(* IEC 61131-3 sources: teller/JD_Teller_LC2_V11/Class/Machine_Settings, 1 file *)

(* ---- Machine_Settings.st ---- *)
(*!
<Class
	Name               = "Machine_Settings"
	Revision           = "1.5"
	RealtimeTask       = "false"
	CyclicTask         = "false"
	BackgroundTask     = "false"
	DefBackground      = "100 ms"
	Sigmatek           = "false"
	OSInterface        = "false"
	HighPriority       = "false"
	Automatic          = "false"
	UpdateMode         = "Prescan"
	SharedCommandTable = "true"
	Objectsize         = "(750,1620)">
	<Channels>
		<Server Name="ClassSvr" Visualized="false" Initialize="false" WriteProtected="true" Retentive="false"/>
		<Server Name="Comp_FreeJam" Visualized="true" Initialize="false" WriteProtected="false" Retentive="false"/>
		<Server Name="Comp_JamTeachIn" Visualized="true" Initialize="false" WriteProtected="false" Retentive="false"/>
		<Server Name="Comp_Teller" Visualized="true" Initialize="false" WriteProtected="false" Retentive="false"/>
		<Server Name="Comp_Teller_Menu" Visualized="true" Initialize="false" WriteProtected="false" Retentive="false"/>
		<Server Name="Comp_Ventieldriver" Visualized="true" Initialize="false" WriteProtected="false" Retentive="false"/>
		<Server Name="Opt_Operator_Login" Visualized="true" Initialize="false" WriteProtected="false" Retentive="false"/>
		<Server Name="Section_View_Rotate" Visualized="true" Initialize="false" WriteProtected="false" Retentive="false"/>
		<Client Name="cComp_FreeJam" Required="false" Internal="false"/>
		<Client Name="cComp_JamTeachIn" Required="false" Internal="false"/>
		<Client Name="cComp_Teller" Required="false" Internal="false"/>
		<Client Name="cComp_Ventieldriver" Required="true" Internal="false"/>
		<Client Name="cOpt_Operator_Login" Required="true" Internal="false"/>
		<Client Name="rComp_Bovenhaak1" Required="true" Internal="true"/>
		<Client Name="rComp_BoxEditor" Required="true" Internal="true"/>
		<Client Name="rComp_Feeder" Required="true" Internal="true"/>
		<Client Name="rComp_FreeJam" Required="true" Internal="true"/>
		<Client Name="rComp_Glue" Required="true" Internal="true"/>
		<Client Name="rComp_Haak1" Required="true" Internal="true"/>
		<Client Name="rComp_Haak2" Required="true" Internal="true"/>
		<Client Name="rComp_Haak3" Required="true" Internal="true"/>
		<Client Name="rComp_JamTeachIn" Required="true" Internal="true"/>
		<Client Name="rComp_RotStop" Required="true" Internal="true"/>
		<Client Name="rComp_Teller" Required="true" Internal="true"/>
		<Client Name="rComp_Ventieldriver" Required="true" Internal="true"/>
		<Client Name="rComp_Voorvouwhaak1" Required="true" Internal="true"/>
		<Client Name="rComp_Voorvouwhaak2" Required="true" Internal="true"/>
		<Client Name="rComp_Vouwriemregeling" Required="true" Internal="true"/>
		<Client Name="rOpt_Operator_Login" Required="true" Internal="true"/>
		<Client Name="rSection_ASection" Required="true" Internal="true"/>
		<Client Name="rSection_BSection" Required="true" Internal="true"/>
		<Client Name="rSection_Conveyor" Required="true" Internal="true"/>
		<Client Name="rSection_CSection" Required="true" Internal="true"/>
		<Client Name="rSection_Feeder" Required="true" Internal="true"/>
		<Client Name="rSection_FinalFold" Required="true" Internal="true"/>
		<Client Name="rSection_FUnit" Required="true" Internal="true"/>
		<Client Name="rSection_MAS" Required="true" Internal="true"/>
		<Client Name="rSection_PreFeeder" Required="true" Internal="true"/>
		<Client Name="rSection_Prefold" Required="true" Internal="true"/>
		<Client Name="rSection_TriFeeder" Required="true" Internal="true"/>
		<Client Name="rSection_Trombone" Required="true" Internal="true"/>
		<Client Name="rSection_View_Rotate" Required="true" Internal="true"/>
	</Channels>
	<RevDoku>
		<Owner Company="JD" Author="JVD"/>
		<Dokumentation Revision="1.5" Date="2014-01-27" Author="JVD" Company="JD" Description="ventieldrivers&#13;&#10;"/>
		<Dokumentation Revision="1.4" Date="2013-06-21" Author="JVD" Company="JD" Description="Extra server voor VVH2 toegevoegd&#13;&#10;"/>
		<Dokumentation Revision="1.3&#13;&#10;" Date="2012-03-28" Author="JVD" Company="JD" Description="Extra server voor de Voorvouwhaak toegevoegd&#13;&#10;"/>
		<Dokumentation Revision="1.2" Date="2011-12-08" Author="JVD" Company="JD" Description="-De servers werden Retentive gemaakt en via SRAM opgeslagen. Af en toe leverde dit problemen op waardoor waarders&#13;&#10;verloren zijn gegaan.&#13;&#10;Dit is opgelost door het gebruikt van Ram classjes in onderliggend netwerk. Peter van Oostrom heeft dit probleem onderkent.&#13;&#10;"/>
		<Dokumentation Revision="1.1" Date="2011-12-06" Author="JVD" Company="JD" Description="De autoSet instellingen zijn toegevoegd"/>
		<Dokumentation Revision="1.0" Date="2011-10-11" Author="JVD" Company="JD" Description="De Server Comp_Freejam toegevoegd"/>
	</RevDoku>
	<Network Name="Machine_Settings">
		<!-- List of Components in this network -->
		<Components>
			<Object
				Name       = "rComp_Bovenhaak1"
				Class      = "Ram"
				Position   = "(180,1620)"
				Visualized = "true">
				<Channels>
					<Server Name="Data"/>
				</Channels>
			</Object>
			<Object
				Name       = "rComp_BoxEditor"
				Class      = "Ram"
				Position   = "(180,180)"
				Visualized = "true">
				<Channels>
					<Server Name="Data"/>
				</Channels>
			</Object>
			<Object
				Name       = "rComp_Feeder"
				Class      = "Ram"
				Position   = "(180,900)"
				Visualized = "true">
				<Channels>
					<Server Name="Data"/>
				</Channels>
			</Object>
			<Object
				Name       = "rComp_FreeJam"
				Class      = "Ram"
				Position   = "(180,1800)"
				Visualized = "true">
				<Channels>
					<Server Name="Data"/>
				</Channels>
			</Object>
			<Object
				Name       = "rComp_Glue"
				Class      = "Ram"
				Position   = "(180,360)"
				Visualized = "true">
				<Channels>
					<Server Name="Data"/>
				</Channels>
			</Object>
			<Object
				Name       = "rComp_Haak1"
				Class      = "Ram"
				Position   = "(180,1080)"
				Visualized = "true">
				<Channels>
					<Server Name="Data"/>
				</Channels>
			</Object>
			<Object
				Name       = "rComp_Haak2"
				Class      = "Ram"
				Position   = "(180,1260)"
				Visualized = "true">
				<Channels>
					<Server Name="Data"/>
				</Channels>
			</Object>
			<Object
				Name       = "rComp_Haak3"
				Class      = "Ram"
				Position   = "(180,1440)"
				Visualized = "true">
				<Channels>
					<Server Name="Data"/>
				</Channels>
			</Object>
			<Object
				Name       = "rComp_JamTeachIn"
				Class      = "Ram"
				Position   = "(600,2160)"
				Visualized = "true">
				<Channels>
					<Server Name="Data"/>
				</Channels>
			</Object>
			<Object
				Name       = "rComp_RotStop"
				Class      = "Ram"
				Position   = "(180,720)"
				Visualized = "true">
				<Channels>
					<Server Name="Data"/>
				</Channels>
			</Object>
			<Object
				Name       = "rComp_Teller"
				Class      = "Ram"
				Position   = "(180,540)"
				Visualized = "true">
				<Channels>
					<Server Name="Data"/>
				</Channels>
			</Object>
			<Object
				Name       = "rComp_Ventieldriver"
				Class      = "Ram"
				Position   = "(180,2520)"
				Visualized = "true">
				<Channels>
					<Server Name="Data"/>
				</Channels>
			</Object>
			<Object
				Name       = "rComp_Voorvouwhaak1"
				Class      = "Ram"
				Position   = "(600,1980)"
				Visualized = "true">
				<Channels>
					<Server Name="Data"/>
				</Channels>
			</Object>
			<Object
				Name       = "rComp_Voorvouwhaak2"
				Class      = "Ram"
				Position   = "(600,2520)"
				Visualized = "true">
				<Channels>
					<Server Name="Data"/>
				</Channels>
			</Object>
			<Object
				Name       = "rComp_Vouwriemregeling"
				Class      = "Ram"
				Position   = "(600,2340)"
				Visualized = "true">
				<Channels>
					<Server Name="Data"/>
				</Channels>
			</Object>
			<Object
				Name       = "rOpt_Operator_Login"
				Class      = "Ram"
				Position   = "(180,2700)"
				Visualized = "true">
				<Channels>
					<Server Name="Data"/>
				</Channels>
			</Object>
			<Object
				Name       = "rSection_ASection"
				Class      = "Ram"
				Position   = "(600,540)"
				Visualized = "true">
				<Channels>
					<Server Name="Data"/>
				</Channels>
			</Object>
			<Object
				Name       = "rSection_BSection"
				Class      = "Ram"
				Position   = "(600,720)"
				Visualized = "true">
				<Channels>
					<Server Name="Data"/>
				</Channels>
			</Object>
			<Object
				Name       = "rSection_Conveyor"
				Class      = "Ram"
				Position   = "(600,1620)"
				Visualized = "true">
				<Channels>
					<Server Name="Data"/>
				</Channels>
			</Object>
			<Object
				Name       = "rSection_CSection"
				Class      = "Ram"
				Position   = "(600,900)"
				Visualized = "true">
				<Channels>
					<Server Name="Data"/>
				</Channels>
			</Object>
			<Object
				Name       = "rSection_Feeder"
				Class      = "Ram"
				Position   = "(180,1980)"
				Visualized = "true">
				<Channels>
					<Server Name="Data"/>
				</Channels>
			</Object>
			<Object
				Name       = "rSection_FinalFold"
				Class      = "Ram"
				Position   = "(600,1080)"
				Visualized = "true">
				<Channels>
					<Server Name="Data"/>
				</Channels>
			</Object>
			<Object
				Name       = "rSection_FUnit"
				Class      = "Ram"
				Position   = "(600,1260)"
				Visualized = "true">
				<Channels>
					<Server Name="Data"/>
				</Channels>
			</Object>
			<Object
				Name       = "rSection_MAS"
				Class      = "Ram"
				Position   = "(600,180)"
				Visualized = "true">
				<Channels>
					<Server Name="Data"/>
				</Channels>
			</Object>
			<Object
				Name       = "rSection_PreFeeder"
				Class      = "Ram"
				Position   = "(180,2160)"
				Visualized = "true">
				<Channels>
					<Server Name="Data"/>
				</Channels>
			</Object>
			<Object
				Name       = "rSection_Prefold"
				Class      = "Ram"
				Position   = "(600,360)"
				Visualized = "true">
				<Channels>
					<Server Name="Data"/>
				</Channels>
			</Object>
			<Object
				Name       = "rSection_TriFeeder"
				Class      = "Ram"
				Position   = "(180,2340)"
				Visualized = "true">
				<Channels>
					<Server Name="Data"/>
				</Channels>
			</Object>
			<Object
				Name       = "rSection_Trombone"
				Class      = "Ram"
				Position   = "(600,1440)"
				Visualized = "true">
				<Channels>
					<Server Name="Data"/>
				</Channels>
			</Object>
			<Object
				Name       = "rSection_View_Rotate"
				Class      = "Ram"
				Position   = "(600,1800)"
				Visualized = "true">
				<Channels>
					<Server Name="Data"/>
				</Channels>
			</Object>
		</Components>
		<Comments>
		</Comments>
		<!-- List of Connections in this network -->
		<Connections>
			<Connection Source="this.rComp_BoxEditor" Destination="rComp_BoxEditor.Data"/>
			<Connection Source="this.rComp_Glue" Destination="rComp_Glue.Data"/>
			<Connection Source="this.rComp_Teller" Destination="rComp_Teller.Data"/>
			<Connection Source="this.rComp_RotStop" Destination="rComp_RotStop.Data"/>
			<Connection Source="this.rComp_Feeder" Destination="rComp_Feeder.Data"/>
			<Connection Source="this.rComp_JamTeachIn" Destination="rComp_JamTeachIn.Data"/>
			<Connection Source="this.rComp_Haak1" Destination="rComp_Haak1.Data"/>
			<Connection Source="this.rComp_Haak2" Destination="rComp_Haak2.Data"/>
			<Connection Source="this.rComp_Haak3" Destination="rComp_Haak3.Data"/>
			<Connection Source="this.rComp_Bovenhaak1" Destination="rComp_Bovenhaak1.Data"/>
			<Connection Source="this.rComp_FreeJam" Destination="rComp_FreeJam.Data"/>
			<Connection Source="this.rSection_Feeder" Destination="rSection_Feeder.Data"/>
			<Connection Source="this.rSection_PreFeeder" Destination="rSection_PreFeeder.Data"/>
			<Connection Source="this.rSection_TriFeeder" Destination="rSection_TriFeeder.Data"/>
			<Connection Source="this.rSection_MAS" Destination="rSection_MAS.Data"/>
			<Connection Source="this.rSection_Prefold" Destination="rSection_Prefold.Data"/>
			<Connection Source="this.rSection_ASection" Destination="rSection_ASection.Data"/>
			<Connection Source="this.rSection_BSection" Destination="rSection_BSection.Data"/>
			<Connection Source="this.rSection_CSection" Destination="rSection_CSection.Data"/>
			<Connection Source="this.rSection_FinalFold" Destination="rSection_FinalFold.Data"/>
			<Connection Source="this.rSection_FUnit" Destination="rSection_FUnit.Data"/>
			<Connection Source="this.rSection_Trombone" Destination="rSection_Trombone.Data"/>
			<Connection Source="this.rSection_Conveyor" Destination="rSection_Conveyor.Data"/>
			<Connection Source="this.rSection_View_Rotate" Destination="rSection_View_Rotate.Data"/>
			<Connection Source="this.rComp_Voorvouwhaak1" Destination="rComp_Voorvouwhaak1.Data"/>
			<Connection Source="this.rComp_Vouwriemregeling" Destination="rComp_Vouwriemregeling.Data"/>
			<Connection Source="this.rComp_Voorvouwhaak2" Destination="rComp_Voorvouwhaak2.Data"/>
			<Connection Source="this.rComp_Ventieldriver" Destination="rComp_Ventieldriver.Data"/>
			<Connection Source="this.rOpt_Operator_Login" Destination="rOpt_Operator_Login.Data"/>
		</Connections>
		<!-- Headerfiles -->
		<Options>
		</Options>
	</Network>
</Class>
*)
Machine_Settings : CLASS
  //Servers:
	ClassSvr 	: SvrChCmd_DINT;
	Comp_Teller_Menu 	: SvrCh_DINT;
	Comp_Teller 	: SvrCh_DINT;
	Comp_Ventieldriver 	: SvrCh_DINT;
	Comp_FreeJam 	: SvrCh_DINT;
	Comp_JamTeachIn 	: SvrCh_DINT;
	Section_View_Rotate 	: SvrCh_DINT;
	Opt_Operator_Login 	: SvrCh_DINT;
  //Clients:
	rComp_BoxEditor 	: CltChCmd_Ram;
	rComp_Glue 	: CltChCmd_Ram;
	rComp_Teller 	: CltChCmd_Ram;
	rComp_RotStop 	: CltChCmd_Ram;
	rComp_Feeder 	: CltChCmd_Ram;
	rComp_Haak1 	: CltChCmd_Ram;
	rComp_Haak2 	: CltChCmd_Ram;
	rComp_Haak3 	: CltChCmd_Ram;
	rComp_Bovenhaak1 	: CltChCmd_Ram;
	rComp_FreeJam 	: CltChCmd_Ram;
	rSection_Feeder 	: CltChCmd_Ram;
	rSection_PreFeeder 	: CltChCmd_Ram;
	rSection_TriFeeder 	: CltChCmd_Ram;
	rSection_MAS 	: CltChCmd_Ram;
	rSection_Prefold 	: CltChCmd_Ram;
	rSection_ASection 	: CltChCmd_Ram;
	rSection_BSection 	: CltChCmd_Ram;
	rSection_CSection 	: CltChCmd_Ram;
	rSection_FinalFold 	: CltChCmd_Ram;
	rSection_FUnit 	: CltChCmd_Ram;
	rSection_Trombone 	: CltChCmd_Ram;
	rSection_Conveyor 	: CltChCmd_Ram;
	rSection_View_Rotate 	: CltChCmd_Ram;
	rComp_Voorvouwhaak1 	: CltChCmd_Ram;
	cComp_Teller 	: CltCh_DINT;
	cComp_Ventieldriver 	: CltCh_DINT;
	cComp_FreeJam 	: CltCh_DINT;
	cComp_JamTeachIn 	: CltCh_DINT;
	cOpt_Operator_Login 	: CltCh_DINT;
	rComp_JamTeachIn 	: CltChCmd_Ram;
	rComp_Vouwriemregeling 	: CltChCmd_Ram;
	rComp_Voorvouwhaak2 	: CltChCmd_Ram;
	rComp_Ventieldriver 	: CltChCmd_Ram;
	rOpt_Operator_Login 	: CltChCmd_Ram;
  //Variables:
  //Functions:

	FUNCTION VIRTUAL GLOBAL Init;

	FUNCTION VIRTUAL GLOBAL Comp_Teller_Menu::Read
		VAR_OUTPUT
			output (EAX) 	: DINT;
		END_VAR;

	FUNCTION VIRTUAL GLOBAL Comp_Teller::Read
		VAR_OUTPUT
			output (EAX) 	: DINT;
		END_VAR;

	FUNCTION VIRTUAL GLOBAL Comp_Teller::Write
		VAR_INPUT
			input (EAX) 	: DINT;
		END_VAR
		VAR_OUTPUT
			result (EAX) 	: DINT;
		END_VAR;

	FUNCTION VIRTUAL GLOBAL Comp_Ventieldriver::Write
		VAR_INPUT
			input (EAX) 	: DINT;
		END_VAR
		VAR_OUTPUT
			result (EAX) 	: DINT;
		END_VAR;

	FUNCTION VIRTUAL GLOBAL Comp_FreeJam::Write
		VAR_INPUT
			input (EAX) 	: DINT;
		END_VAR
		VAR_OUTPUT
			result (EAX) 	: DINT;
		END_VAR;

	FUNCTION VIRTUAL GLOBAL Comp_JamTeachIn::Write
		VAR_INPUT
			input (EAX) 	: DINT;
		END_VAR
		VAR_OUTPUT
			result (EAX) 	: DINT;
		END_VAR;

	FUNCTION VIRTUAL GLOBAL Section_View_Rotate::Write
		VAR_INPUT
			input (EAX) 	: DINT;
		END_VAR
		VAR_OUTPUT
			result (EAX) 	: DINT;
		END_VAR;

	FUNCTION VIRTUAL GLOBAL Opt_Operator_Login::Write
		VAR_INPUT
			input (EAX) 	: DINT;
		END_VAR
		VAR_OUTPUT
			result (EAX) 	: DINT;
		END_VAR;
  //Tables:
	FUNCTION @STD
		VAR_OUTPUT
			ret_code	: CONFSTATES;
		END_VAR;
	FUNCTION GLOBAL TAB @CT_;
END_CLASS;

#pragma using Ram

FUNCTION VIRTUAL GLOBAL Machine_Settings::Init

    if    _FirstScan then

          rComp_Teller := rComp_Teller.Read();
          rComp_Ventieldriver := rComp_Ventieldriver.Read();
          rComp_FreeJam := rComp_FreeJam.Read();
          rComp_JamTeachIn := rComp_JamTeachIn.Read();
          rOpt_Operator_Login := rOpt_Operator_Login.Read();

          Comp_Teller.Write(input:=rComp_Teller);
          Comp_Ventieldriver.Write(input:=rComp_Ventieldriver);
          Comp_FreeJam.Write(input:=rComp_FreeJam);
          Comp_JamTeachIn.Write(input:=rComp_JamTeachIn);
          Opt_Operator_Login.Write(input:=rOpt_Operator_Login);
          Comp_Teller := 1;
          cComp_Teller.Write(Comp_Teller);

    end_if;

END_FUNCTION

FUNCTION VIRTUAL GLOBAL Machine_Settings::Comp_Teller::Write
	VAR_INPUT
		input (EAX) 	: DINT;
	END_VAR
	VAR_OUTPUT
		result (EAX) 	: DINT;
	END_VAR

	Comp_Teller := input;
  rComp_Teller.Write(input:=Comp_Teller);
  cComp_Teller := Comp_Teller;
  cComp_Teller.Write(input:=Comp_Teller);
 	result := Comp_Teller;

END_FUNCTION

FUNCTION VIRTUAL GLOBAL Machine_Settings::Comp_FreeJam::Write
	VAR_INPUT
		input (EAX) 	: DINT;
	END_VAR
	VAR_OUTPUT
		result (EAX) 	: DINT;
	END_VAR

	Comp_FreeJam := input;
  rComp_FreeJam.Write(input:=Comp_FreeJam);
  cComp_FreeJam := Comp_FreeJam;
  cComp_FreeJam.Write(input:=Comp_FreeJam);
 	result := Comp_FreeJam;

END_FUNCTION

FUNCTION VIRTUAL GLOBAL Machine_Settings::Section_View_Rotate::Write
	VAR_INPUT
		input (EAX) 	: DINT;
	END_VAR
	VAR_OUTPUT
		result (EAX) 	: DINT;
	END_VAR

	Section_View_Rotate := input;
  rSection_View_Rotate.Write(input:=Section_View_Rotate);
 	result := Section_View_Rotate;

END_FUNCTION

FUNCTION VIRTUAL GLOBAL Machine_Settings::Comp_JamTeachIn::Write
	VAR_INPUT
		input (EAX) 	: DINT;
	END_VAR
	VAR_OUTPUT
		result (EAX) 	: DINT;
	END_VAR

	Comp_JamTeachIn := input;
  rComp_JamTeachIn.Write(input:=Comp_JamTeachIn);
  cComp_JamTeachIn := Comp_JamTeachIn;
  cComp_JamTeachIn.Write(input:=Comp_JamTeachIn);
 	result := Comp_JamTeachIn;

END_FUNCTION

FUNCTION VIRTUAL GLOBAL Machine_Settings::Comp_Ventieldriver::Write
	VAR_INPUT
		input (EAX) 	: DINT;
	END_VAR
	VAR_OUTPUT
		result (EAX) 	: DINT;
	END_VAR

	Comp_Ventieldriver := input;
  rComp_Ventieldriver.Write(input:=Comp_Ventieldriver);
  cComp_Ventieldriver := Comp_Ventieldriver;
  cComp_Ventieldriver.Write(input:=Comp_Ventieldriver);
	result := Comp_Ventieldriver;

END_FUNCTION

FUNCTION VIRTUAL GLOBAL Machine_Settings::Comp_Teller_Menu::Read
	VAR_OUTPUT
		output (EAX) 	: DINT;
	END_VAR

  // Menuknop vouwhaken enkel weergeven als er tenminste 1 type haak in gebruik is
  if Comp_Teller or Comp_Ventieldriver then
    Comp_Teller_Menu :=1;
  else
    Comp_Teller_Menu :=0;
  end_if;
	output := Comp_Teller_Menu;

END_FUNCTION

FUNCTION VIRTUAL GLOBAL Machine_Settings::Opt_Operator_Login::Write
	VAR_INPUT
		input (EAX) 	: DINT;
	END_VAR
	VAR_OUTPUT
		result (EAX) 	: DINT;
	END_VAR

	Opt_Operator_Login := input;
  rOpt_Operator_Login.Write(input:=Opt_Operator_Login);
  cOpt_Operator_Login := Opt_Operator_Login;
  cOpt_Operator_Login.Write(input:=Opt_Operator_Login);
	result := Opt_Operator_Login;

END_FUNCTION

FUNCTION VIRTUAL GLOBAL Machine_Settings::Comp_Teller::Read
	VAR_OUTPUT
		output (EAX) 	: DINT;
	END_VAR

  // aanpassing 20140730 DW
  Comp_Teller := 1;
  cComp_Teller.Write(Comp_Teller);
	output := Comp_Teller;

END_FUNCTION
